(* IEC 61131-3 sources: POMIRTS_lab3/AS/Library_2/ArEco, 3 files *)

(* ---- ArEco.typ ---- *)
TYPE
	ArEcoWakeupModeEnum :
		( (*Wake-up mode*)
		arECO_WAKEUPMODE_DISABLED := 0, (*Disable the wake-up trigger*)
		arECO_WAKEUPMODE_VISIBLE := 1, (*Wake-up visible: Turn on display and LEDs*)
		arECO_WAKEUPMODE_SILENT := 2 (*Wake-up silent: Turn off display and LEDs*)
		);
	ArEcoWakeupTriggerType : 	STRUCT  (*Wake-up trigger parameters*)
		Name : STRING[80]; (*Name of the wake-up trigger*)
		Mode : ArEcoWakeupModeEnum; (*Wake-up mode*)
	END_STRUCT;
	ArEcoWakeupTimeType : 	STRUCT  (*Wake-up time parameters*)
		Time : TIME; (*Target time for wake-up*)
		Mode : ArEcoWakeupModeEnum; (*Wake-up mode*)
	END_STRUCT;
END_TYPE

(* ---- ArEco.fun ---- *)
{REDUND_ERROR} {REDUND_UNREPLICABLE} FUNCTION_BLOCK ArEcoPlcShutdown (*Select wake-up triggers and shutdown the PLC; asynchronous execution*)
	VAR_INPUT
		Execute : BOOL; (*Start execution*)
		WakeupTriggers : REFERENCE TO ArEcoWakeupTriggerType; (*Array of wake-up triggers*)
		NrOfWakeupTriggers : UINT; (*Number of wake-up triggers in array*)
		WakeupTime : ArEcoWakeupTimeType; (*Target time for wake-up*)
	END_VAR
	VAR_OUTPUT
		Done : BOOL; (*Execution successful*)
		Busy : BOOL; (*Execution running*)
		Error : BOOL; (*Execution failed*)
		StatusID : DINT; (*Execution status information: see help*)
		InvalidWakeupTrigger : STRING[80]; (*Name of the wrong wake-up trigger*)
	END_VAR
	VAR
		Internal : ARRAY[0..31] OF UDINT;
	END_VAR
END_FUNCTION_BLOCK

{REDUND_ERROR} {REDUND_UNREPLICABLE} FUNCTION_BLOCK ArEcoPlcWakeupInfo (*Get PLC wake-up information; asynchronous execution*)
	VAR_INPUT
		Execute : BOOL; (*Start execution*)
	END_VAR
	VAR_OUTPUT
		Done : BOOL; (*Execution successful*)
		Busy : BOOL; (*Execution running*)
		Error : BOOL; (*Execution failed*)
		StatusID : DINT; (*Execution status information: see help*)
		TriggeredWakeup : BOOL; (*A wake-up trigger has triggered*)
		TimedWakeup : BOOL; (*Wake-up time has triggered*)
		SilentWakeup : BOOL; (*The wake-up was silent: Display and LEDs are switched off*)
	END_VAR
	VAR
		Internal : ARRAY[0..31] OF UDINT;
	END_VAR
END_FUNCTION_BLOCK

{REDUND_ERROR} {REDUND_UNREPLICABLE} FUNCTION_BLOCK ArEcoPlcWakeupTriggerState (*Get the state of a specified wake-up trigger; asynchronous execution*)
	VAR_INPUT
		Execute : BOOL; (*Start execution*)
		Name : STRING[80]; (*Name of the wake-up trigger*)
	END_VAR
	VAR_OUTPUT
		Done : BOOL; (*Execution successful*)
		Busy : BOOL; (*Execution running*)
		Error : BOOL; (*Execution failed*)
		StatusID : DINT; (*Execution status information: see help*)
		Triggered : BOOL; (*The wake-up trigger has triggered*)
	END_VAR
	VAR
		Internal : ARRAY[0..31] OF UDINT;
	END_VAR
END_FUNCTION_BLOCK

(* ---- ArEco.var ---- *)
VAR CONSTANT
	arECO_ERR_FB_NOT_SUPPORTED : DINT := -1070584446; (*The used PLC do not support this functionblock*)
	arECO_ERR_INVALID_PARAMETER : DINT := -1070584445; (*Please check function block parameters*)
	arECO_ERR_INTERNAL : DINT := -1070584444; (*An internal error has occurred: Please contact B+R support*)
	arECO_ERR_INVALID_WAKEUPTRIGGER : DINT := -1070584443; (*Please check wake-up triggers*)
	arECO_ERR_INVALID_WAKEUPMODE : DINT := -1070584442; (*Please check wake-up modes*)
	arECO_ERR_NO_WAKEUP_PAR : DINT := -1070584441; (*No wake-up parameters set*)
END_VAR
